// TIA Portal project "Abfüllanlage" (V15)

(* hardware
DEVICE "S7-1200-Station_1"  S7-1200 Station
   slot 0: "Baugruppenträger_0"  S7-1200 Rack  Rack  V1.0
   slot 1: "PLC_1"  CPU 1214C DC/DC/Rly  6ES7 214-1HG40-0XB0  V4.2
*)

// ===== PLC "PLC_1"  CPU 1214C DC/DC/Rly =====

VAR_GLOBAL   // PLC tag table "Standard-Variablentabelle"
   "Clock_Byte" AT %MB100 : Byte;
   "Clock_10Hz" AT %M100.0 : Bool;
   "Clock_5Hz" AT %M100.1 : Bool;
   "Clock_2.5Hz" AT %M100.2 : Bool;
   "Clock_2Hz" AT %M100.3 : Bool;
   "Clock_1.25Hz" AT %M100.4 : Bool;
   "Clock_1Hz" AT %M100.5 : Bool;
   "Clock_0.625Hz" AT %M100.6 : Bool;
   "Clock_0.5Hz" AT %M100.7 : Bool;
   "S1" AT %I0.0 : Bool;   // Anlage Start
   "S2" AT %I0.1 : Bool;   // Anlage Stop
   "S3" AT %I0.2 : Bool;   // Vereinzelung
   "S4" AT %I0.3 : Bool;   // Quittieren
   "F5" AT %I0.4 : Bool;   // Motorschutzschalter
   "B1" AT %I0.5 : Bool;   // Sensor Flasche
   "P1" AT %Q0.0 : Bool;   // Anlage Ein
   "P2" AT %Q0.1 : Bool;   // Anlage Störung
   "Q1" AT %Q0.2 : Bool;   // Motor Förderband
   "K1" AT %Q0.3 : Bool;   // Füllventil Flasche
   "K2" AT %Q0.4 : Bool;   // Ventil Vereinzelung Flasche
   "Merker Betriebsbereit" AT %M10.0 : Bool;   // Betriebsbereit
   "Merker Sammelstörung" AT %M10.1 : Bool;
   "Füllstand AI" AT %IW64 : Word;
   "Zyklus Start" AT %M10.2 : Bool;
   "Vereinzelung Schritt1" AT %M10.3 : Bool;
   "Förderband Schritt2" AT %M10.4 : Bool;
   "Füllung Schritt3" AT %M10.5 : Bool;
   "Förderband Schritt4" AT %M10.6 : Bool;
   "Zyklus Ende" AT %M10.7 : Bool;
   "Merker Störung MSS" AT %M11.0 : Bool;
   "Merker Störung Vereinzeln" AT %M11.1 : Bool;
   "Merker Störung Füllung" AT %M11.2 : Bool;
END_VAR

DATA_BLOCK "Analogwertverarbeitung"   // DB3
{ S7_Optimized_Access := 'TRUE' }
VERSION : 0.1
   VAR
      "Analogwert Normieren" : Int;
      "Analogwert Skalieren" : Real;
   END_VAR
BEGIN
END_DATA_BLOCK

// folder: System blocks/Program resources

DATA_BLOCK "IEC_Timer_0_DB"   // DB1
{ S7_Optimized_Access := 'TRUE' }
AUTHOR : Simatic
FAMILY : IEC
NAME : IEC_TMR
VERSION : 1.0
// stored: InstanceOfName IEC_TIMER
"IEC_TIMER"
BEGIN
END_DATA_BLOCK

DATA_BLOCK "IEC_Timer_0_DB_1"   // DB2
{ S7_Optimized_Access := 'TRUE' }
AUTHOR : Simatic
FAMILY : IEC
NAME : IEC_TMR
VERSION : 1.0
// stored: InstanceOfName IEC_TIMER
"IEC_TIMER"
BEGIN
END_DATA_BLOCK

DATA_BLOCK "IEC_Timer_0_DB_2"   // DB4
{ S7_Optimized_Access := 'TRUE' }
AUTHOR : Simatic
FAMILY : IEC
NAME : IEC_TMR
VERSION : 1.0
// stored: InstanceOfName IEC_TIMER
"IEC_TIMER"
BEGIN
END_DATA_BLOCK

DATA_BLOCK "IEC_Timer_0_DB_3"   // DB5
{ S7_Optimized_Access := 'TRUE' }
AUTHOR : Simatic
FAMILY : IEC
NAME : IEC_TMR
VERSION : 1.0
// stored: InstanceOfName IEC_TIMER
"IEC_TIMER"
BEGIN
END_DATA_BLOCK

DATA_BLOCK "IEC_Timer_0_DB_4"   // DB6
{ S7_Optimized_Access := 'TRUE' }
AUTHOR : Simatic
FAMILY : IEC
NAME : IEC_TMR
VERSION : 1.0
// stored: InstanceOfName IEC_TIMER
"IEC_TIMER"
BEGIN
END_DATA_BLOCK

DATA_BLOCK "IEC_Timer_0_DB_5"   // DB7
{ S7_Optimized_Access := 'TRUE' }
AUTHOR : Simatic
FAMILY : IEC
NAME : IEC_TMR
VERSION : 1.0
// stored: InstanceOfName IEC_TIMER
"IEC_TIMER"
BEGIN
END_DATA_BLOCK

DATA_BLOCK "IEC_Timer_0_DB_6"   // DB8
{ S7_Optimized_Access := 'TRUE' }
AUTHOR : Simatic
FAMILY : IEC
NAME : IEC_TMR
VERSION : 1.0
// stored: InstanceOfName IEC_TIMER
"IEC_TIMER"
BEGIN
END_DATA_BLOCK

DATA_BLOCK "IEC_Timer_0_DB_7"   // DB9
{ S7_Optimized_Access := 'TRUE' }
AUTHOR : Simatic
FAMILY : IEC
NAME : IEC_TMR
VERSION : 1.0
// stored: InstanceOfName IEC_TIMER
"IEC_TIMER"
BEGIN
END_DATA_BLOCK

DATA_BLOCK "IEC_Timer_0_DB_8"   // DB10
{ S7_Optimized_Access := 'TRUE' }
AUTHOR : Simatic
FAMILY : IEC
NAME : IEC_TMR
VERSION : 1.0
// stored: InstanceOfName IEC_TIMER
"IEC_TIMER"
BEGIN
END_DATA_BLOCK

DATA_BLOCK "IEC_Timer_0_DB_9"   // DB11
{ S7_Optimized_Access := 'TRUE' }
AUTHOR : Simatic
FAMILY : IEC
NAME : IEC_TMR
VERSION : 1.0
// stored: InstanceOfName IEC_TIMER
"IEC_TIMER"
BEGIN
END_DATA_BLOCK

// folder: (top level)

FUNCTION "Abfüllanlage" : Void   // FC1, FBD
TITLE = Abfüllanlage
{ S7_Optimized_Access := 'TRUE' }
VERSION : 0.1
BEGIN

REGION Network 1: Anlage Ein
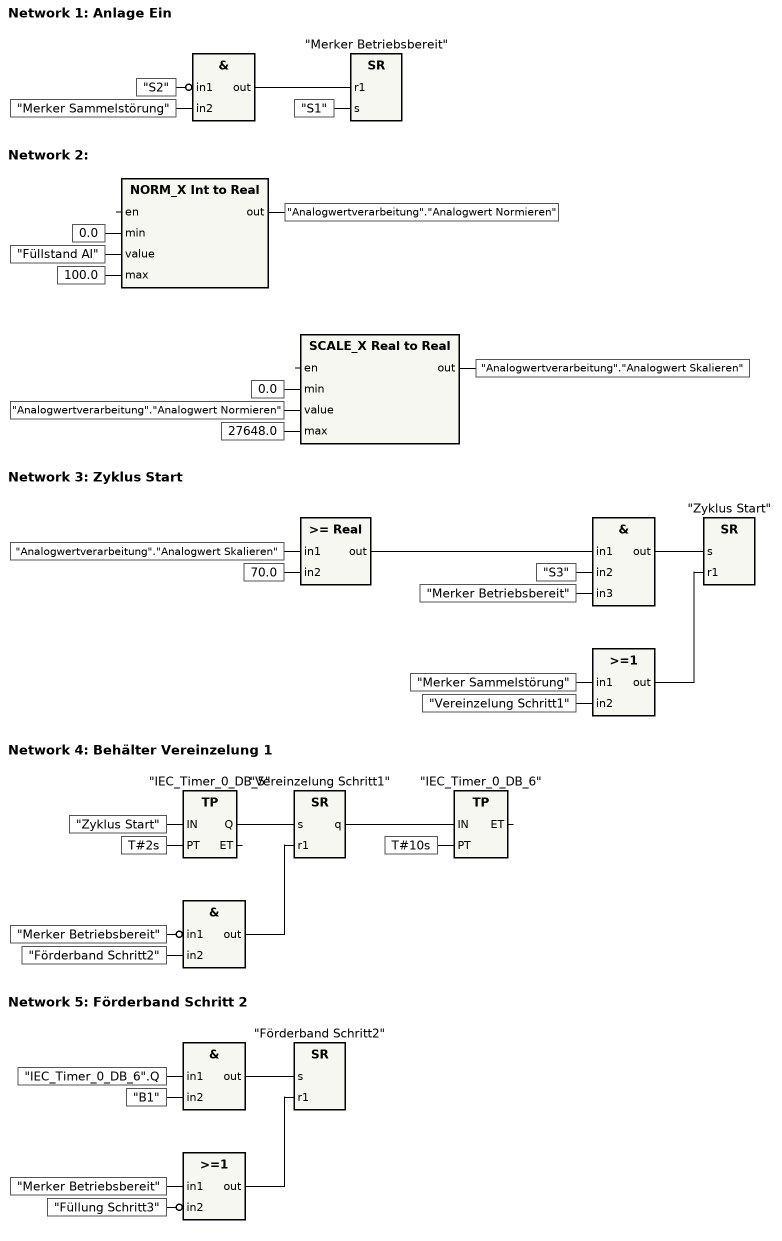
   IF "S1" THEN
       "Merker Betriebsbereit" := TRUE;   // SR flip-flop
   END_IF;
   IF NOT "S2" AND "Merker Sammelstörung" THEN "Merker Betriebsbereit" := FALSE; END_IF;
END_REGION

REGION Network 2
   "Analogwertverarbeitung"."Analogwert Normieren" := NORM_X(MIN := 0.0, VALUE := "Füllstand AI", MAX := 100.0);
   "Analogwertverarbeitung"."Analogwert Skalieren" := SCALE_X(MIN := 0.0, VALUE := "Analogwertverarbeitung"."Analogwert Normieren", MAX := 27648.0);
END_REGION

REGION Network 3: Zyklus Start
   IF ("Analogwertverarbeitung"."Analogwert Skalieren" >= 70.0) AND "S3" AND "Merker Betriebsbereit" THEN
       "Zyklus Start" := TRUE;   // SR flip-flop
   END_IF;
   IF "Merker Sammelstörung" OR "Vereinzelung Schritt1" THEN "Zyklus Start" := FALSE; END_IF;
END_REGION

REGION Network 4: Behälter Vereinzelung 1
   "IEC_Timer_0_DB_5".TP(IN := "Zyklus Start", PT := T#2s);
   IF "IEC_Timer_0_DB_5".Q THEN
       "Vereinzelung Schritt1" := TRUE;   // SR flip-flop
   END_IF;
   IF NOT "Merker Betriebsbereit" AND "Förderband Schritt2" THEN "Vereinzelung Schritt1" := FALSE; END_IF;
   "IEC_Timer_0_DB_6".TP(IN := "Vereinzelung Schritt1", PT := T#10s);
END_REGION

REGION Network 5: Förderband Schritt 2
   IF "IEC_Timer_0_DB_6".Q AND "B1" THEN
       "Förderband Schritt2" := TRUE;   // SR flip-flop
   END_IF;
   IF "Merker Betriebsbereit" OR NOT "Füllung Schritt3" THEN "Förderband Schritt2" := FALSE; END_IF;
END_REGION

REGION Network 6: Füllung
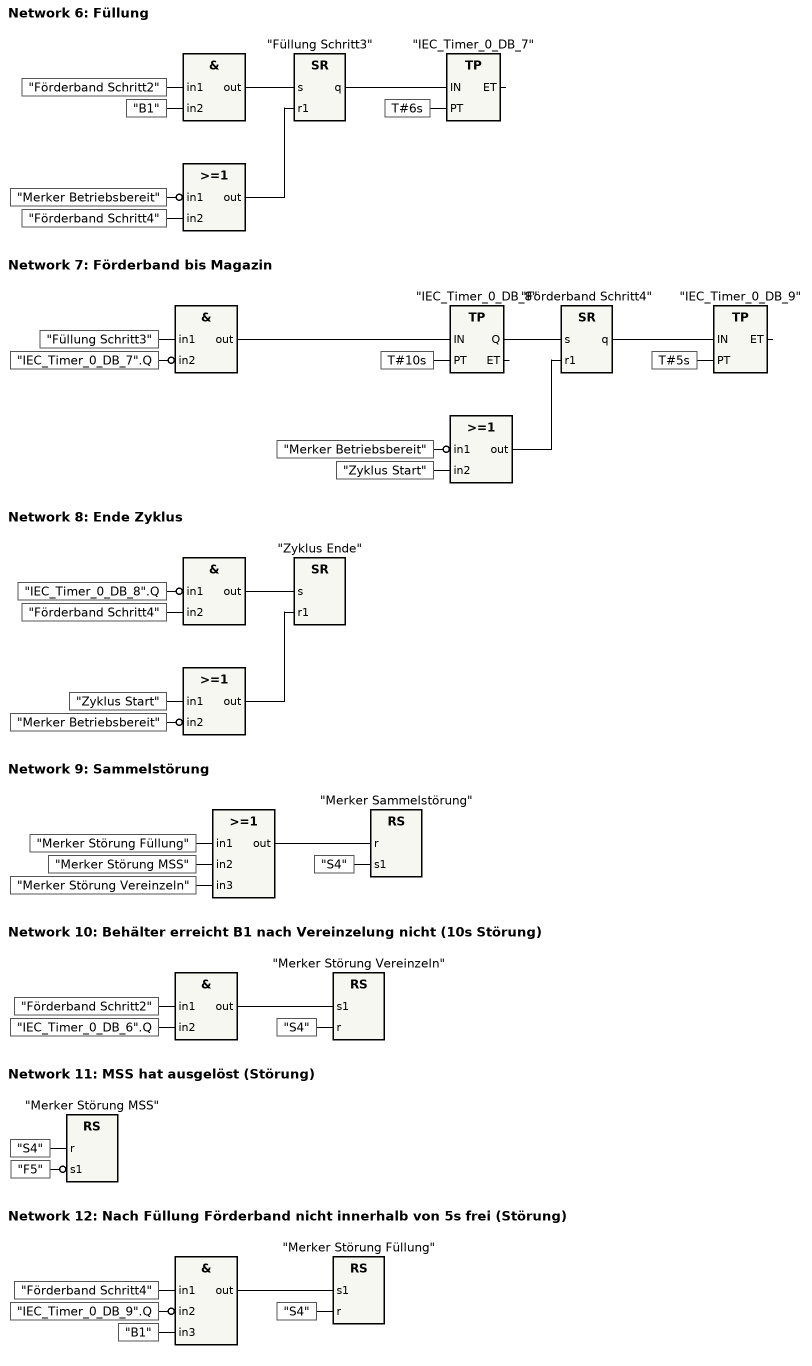
   IF "Förderband Schritt2" AND "B1" THEN
       "Füllung Schritt3" := TRUE;   // SR flip-flop
   END_IF;
   IF NOT "Merker Betriebsbereit" OR "Förderband Schritt4" THEN "Füllung Schritt3" := FALSE; END_IF;
   "IEC_Timer_0_DB_7".TP(IN := "Füllung Schritt3", PT := T#6s);
END_REGION

REGION Network 7: Förderband bis Magazin
   "IEC_Timer_0_DB_8".TP(IN := "Füllung Schritt3" AND NOT "IEC_Timer_0_DB_7".Q, PT := T#10s);
   IF "IEC_Timer_0_DB_8".Q THEN
       "Förderband Schritt4" := TRUE;   // SR flip-flop
   END_IF;
   IF NOT "Merker Betriebsbereit" OR "Zyklus Start" THEN "Förderband Schritt4" := FALSE; END_IF;
   "IEC_Timer_0_DB_9".TP(IN := "Förderband Schritt4", PT := T#5s);
END_REGION

REGION Network 8: Ende Zyklus
   IF NOT "IEC_Timer_0_DB_8".Q AND "Förderband Schritt4" THEN
       "Zyklus Ende" := TRUE;   // SR flip-flop
   END_IF;
   IF "Zyklus Start" OR NOT "Merker Betriebsbereit" THEN "Zyklus Ende" := FALSE; END_IF;
END_REGION

REGION Network 9: Sammelstörung
   IF "Merker Störung Füllung" OR "Merker Störung MSS" OR "Merker Störung Vereinzeln" THEN
       "Merker Sammelstörung" := FALSE;   // RS flip-flop
   END_IF;
   IF "S4" THEN "Merker Sammelstörung" := TRUE; END_IF;
END_REGION

REGION Network 10: Behälter erreicht B1 nach Vereinzelung nicht (10s Störung)
   IF "S4" THEN
       "Merker Störung Vereinzeln" := FALSE;   // RS flip-flop
   END_IF;
   IF "Förderband Schritt2" AND "IEC_Timer_0_DB_6".Q THEN "Merker Störung Vereinzeln" := TRUE; END_IF;
END_REGION

REGION Network 11: MSS hat ausgelöst (Störung)
   IF "S4" THEN
       "Merker Störung MSS" := FALSE;   // RS flip-flop
   END_IF;
   IF NOT "F5" THEN "Merker Störung MSS" := TRUE; END_IF;
END_REGION

REGION Network 12: Nach Füllung Förderband nicht innerhalb von 5s frei (Störung)
   IF "S4" THEN
       "Merker Störung Füllung" := FALSE;   // RS flip-flop
   END_IF;
   IF "Förderband Schritt4" AND NOT "IEC_Timer_0_DB_9".Q AND "B1" THEN
       "Merker Störung Füllung" := TRUE;
   END_IF;
END_REGION

REGION Network 13: Motorschütz M1
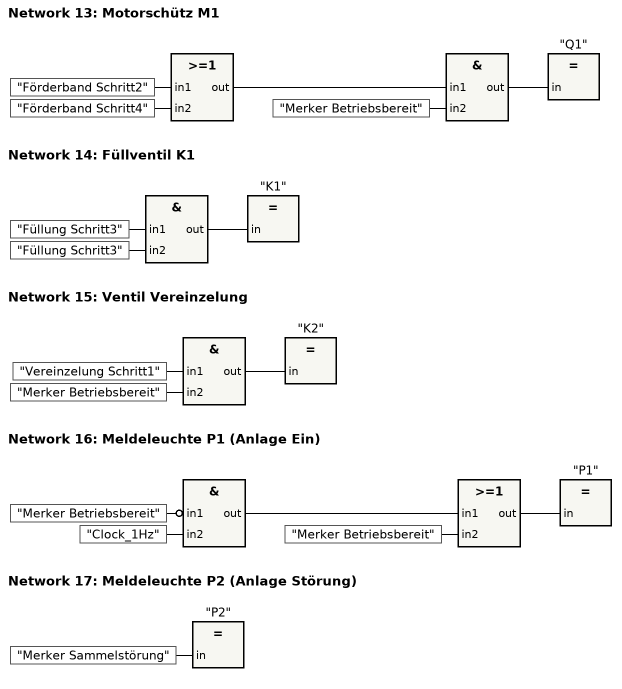
   "Q1" := ("Förderband Schritt2" OR "Förderband Schritt4") AND "Merker Betriebsbereit";
END_REGION

REGION Network 14: Füllventil K1
   "K1" := "Füllung Schritt3" AND "Füllung Schritt3";
END_REGION

REGION Network 15: Ventil Vereinzelung
   "K2" := "Vereinzelung Schritt1" AND "Merker Betriebsbereit";
END_REGION

REGION Network 16: Meldeleuchte P1 (Anlage Ein)
   "P1" := (NOT "Merker Betriebsbereit" AND "Clock_1Hz") OR "Merker Betriebsbereit";
END_REGION

REGION Network 17: Meldeleuchte P2 (Anlage Störung)
   "P2" := "Merker Sammelstörung";
END_REGION
END_FUNCTION

ORGANIZATION_BLOCK "Main"   // OB1, LAD, ProgramCycle
TITLE = "Main Program Sweep (Cycle)"
{ S7_Optimized_Access := 'TRUE' }
VERSION : 0.1
   VAR_INPUT
      Initial_Call : Bool;   // Initial call of this OB
      Remanence : Bool;   // =True, if remanent data are available
   END_VAR
BEGIN

REGION Network 1
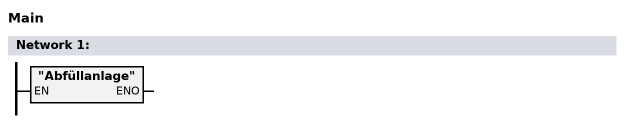
   RUNG wire#powerrail
      "Abfüllanlage"()
   END_RUNG
   // the same network as SCL:
   "Abfüllanlage"();
END_REGION
END_ORGANIZATION_BLOCK